PROGRAM MAIN
VAR
	VTD : VTD_FB;
END_VAR

VTD.

END_PROGRAM

(* stored: Version 1.1.0.1
   POU MAIN: Id {1668c7a5-c10d-4b27-a3e5-4fc8521ffe20}, SpecialFunc None *)
